(* PLC project Untitled1, Beckhoff Automation GmbH TwinCAT PLC Control 3.5.13.20 *)
(* stored: creationDateTime 2022-07-20T15:22:49.2677045, modificationDateTime 2022-07-20T15:22:49.2677045 *)

{attribute 'qualified_only'}
{attribute 'strict'}
TYPE eFirmerEvent : (eNoInfo := 0, eGroundFault := 1, eDCOverVolt := 2, eACDisconnect := 3, eDCDisconnect := 4, eGridDisconnect := 5, eCabinetOpen := 6, eManualShutdown := 7, eOverTemp := 8, eOverFrequency := 9, eUnderFrequency := 10, eACOverVolt := 11, eACUnderVolt := 12, eBlownStringFuse := 13, eUnderTemp := 14, eMemoryLoss := 15, eHWTestFailure := 16);
END_TYPE
